TEXTLIST ModeStatesHeader
  0 = 'No State' | 汉语: '汉语'
  1 = 'Power Off' | 汉语: '汉语'
  2 = 'Power On' | 汉语: '汉语'
  3 = 'Manual' | 汉语: '汉语'
  4 = 'Auto'
  5 = 'Auto Cycle'
  6 = 'Semi Auto'
  7 = 'Fault'
  8 = 'Bypass'
  9 = 'Stopping'
  10 = 'State2'
   = ''
END_TEXTLIST

(* stored: Version 1.1.0.1, ProductVersion 3.1.4024.11
   TextList ModeStatesHeader: Id {034afc55-d990-4fdc-a4bf-a6c19d18859f} *)
